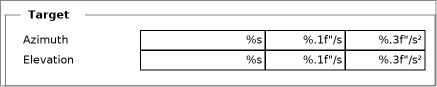
VISUALIZATION VISU_AxesFromCpp_Target  // 437x87
VAR_IN_OUT
	ref : Axes;
    widget : AxesWidget;
END_VAR
    Polyline (20,15) (5,15) (5,85) (435,85) (435,15) (85,15)
    Label (25,5 60x20), "Target"
    Label (20,30 80x20), "Azimuth"
    Label (20,50 80x20), "Elevation"
    Rectangle (140,30 125x20), "%s", text variable: widget.axes.azi.targetPos.dmsString
    Rectangle (140,50 125x20), "%s", text variable: widget.axes.ele.targetPos.dmsString
    Rectangle (265,30 80x20), "%.1f"/s", text variable: ref.target.aziVelo.arcsecondsPerSecond.value
    Rectangle (345,30 80x20), "%.3f"/s²", text variable: ref.target.aziAcc.arcsecondsPerSquareSecond.value
    Rectangle (345,50 80x20), "%.3f"/s²", text variable: ref.target.eleAcc.arcsecondsPerSquareSecond.value
    Rectangle (265,50 80x20), "%.1f"/s", text variable: ref.target.eleVelo.arcsecondsPerSecond.value
END_VISUALIZATION

(* stored: Version 1.1.0.1, ProductVersion 3.1.4019.2
   Visu VISU_AxesFromCpp_Target: Id {63b9ca13-e736-4c35-925b-556e4f0fc3d8} *)
